# EPICS substitutions: iocs/MC12/tpmacApp/Db/pmacStatus.substitutions
file "db/pmacStatus.db"
{
pattern
{SYS,            PMAC,    VERSION  PLC  PORT,  NAXES }
{"XF:06BM-CT",   "MC:12", "1"      5    "P0",  8     }
}
